// Core §8.13 — semantic HAL output; a project Hardware Driver owns channel maps.
TYPE ST_SignalTowerOut :
STRUCT
    Red      : BOOL;
    Amber    : BOOL;
    Green    : BOOL;
    Blue     : BOOL;
    White    : BOOL;
    Horn     : BOOL;
    TestActive : BOOL;
END_STRUCT
END_TYPE

(* stored: Version 1.1.0.1, ProductVersion 3.1.4024.12
   DUT ST_SignalTowerOut: Id {d0c37f12-27ee-4653-9a95-7d12c8e1164f} *)
